# EPICS substitutions: pimegaApp/Db/pimega135d.substitutions
file "module.template" {
   pattern { MODULE, ADDR }
           { M1:,    0    }
}
